FUNCTION_BLOCK FB_Motion1way
VAR

	tIsAdvancReq: BOOL;
	timOnDelay: TON;

END_VAR

VAR_INPUT
	iAdvanceReq: BOOL;
	iAdvanced: BOOL;
	iTimeoutVal:TIME := T#5S;
	iMode: typeStationMode; //what mode is station in?
END_VAR
VAR_OUTPUT
	qAdvanceFault: BOOL;
	qIsAdvancing: BOOL;

END_VAR
VAR // added by the converter: edge detectors and wires of the graphical bodies
    _rt1 : R_TRIG;
END_VAR

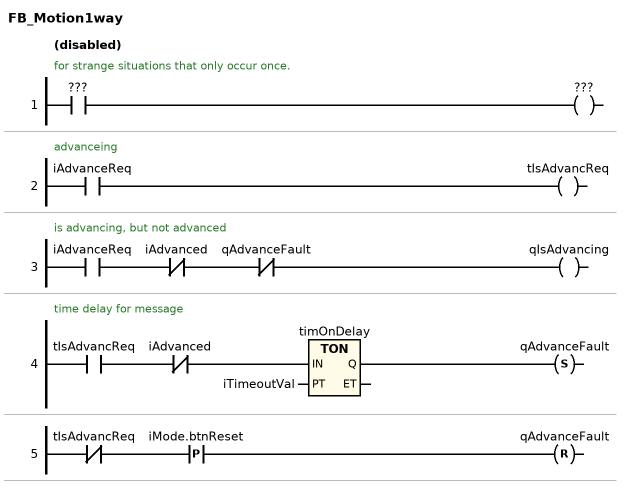
// NETWORK 1 (disabled)
// for strange situations that only occur once.
// ??? := ???;

// NETWORK 2
// advanceing
tIsAdvancReq := iAdvanceReq;

// NETWORK 3
// is advancing, but not advanced
qIsAdvancing := iAdvanceReq AND NOT iAdvanced AND NOT qAdvanceFault;

// NETWORK 4
// time delay for message
timOnDelay(IN := tIsAdvancReq AND NOT iAdvanced, PT := iTimeoutVal); // TON
qAdvanceFault S= timOnDelay.Q;

// NETWORK 5
_rt1(CLK := iMode.btnReset);
qAdvanceFault R= NOT tIsAdvancReq AND _rt1.Q;

END_FUNCTION_BLOCK

(* stored: Version 1.1.0.1, ProductVersion 3.1.4024.12
   POU FB_Motion1way: Id {94bc97ff-8896-4204-82e1-db7f8bcefc22}, SpecialFunc None *)
